(* CoDeSys 2.3 export: EDGEDETECTION.EXP *)

(* POU Components/EdgeDetection, ST *)
FUNCTION_BLOCK EdgeDetection
VAR_INPUT
	input:BOOL;
END_VAR
VAR_OUTPUT
	output: BOOL;
END_VAR
VAR
	oldValue: BOOL;
	onFallingEdge:BOOL := 1;
END_VAR
VAR_IN_OUT
END_VAR
IF onFallingEdge THEN
	output:= (oldValue = 1) AND (input = 0);
ELSE
	output:= (oldValue = 0) AND (input = 1);
END_IF
oldValue:= input;
END_FUNCTION_BLOCK
